FUNCTION_BLOCK AUS_FIELDBUS_USINT_TO_SIGNAL_SCALED (* Mirrors IN->OUT if Signal Valid, with scaling *)
  (* Standard: 61499-1; Description: Copyright (c) 2026 HR Agrartechnik GmbH This program and the accompanying materials are made available under the terms of the Eclipse Public License 2.0 which is available at https://www.eclipse.org/legal/epl-2.0/ SPDX-License-Identifier: EPL-2.0 *)
  (* Version 1.0, 2026-05-31, Franz Höpfinger, HR Agrartechnik GmbH *)
  PACKAGE logiBUS::signalprocessing::fieldbus;
  IMPORT eclipse4diac::core::TypeHash;
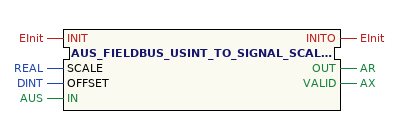
  EVENT_INPUT
    INIT : EInit; (* Init Request *)
  END_EVENT
  EVENT_OUTPUT
    INITO : EInit; (* Init Confirmation *)
  END_EVENT
  VAR_INPUT
    SCALE : REAL := REAL#1.0; (* Scaling factor *)
    OFFSET : DINT := DINT#0; (* Offset added after scaling *)
  END_VAR
  SOCKETS
    IN : adapter::types::unidirectional::AUS; (* Input *)
  END_SOCKETS
  PLUGS
    OUT : adapter::types::unidirectional::AR; (* Output Filtered *)
    VALID : adapter::types::unidirectional::AX; (* TRUE if Signal is VALID *)
  END_PLUGS
  FBS
    FIELDBUS_USINT_TO_SIGNAL_SCALED : logiBUS::signalprocessing::fieldbus::FIELDBUS_USINT_TO_SIGNAL_SCALED;
    E_D_FF : iec61499::events::E_D_FF;
  END_FBS
  EVENT_CONNECTIONS
    IN.E1 TO FIELDBUS_USINT_TO_SIGNAL_SCALED.REQ;
    FIELDBUS_USINT_TO_SIGNAL_SCALED.CNF TO OUT.E1;
    FIELDBUS_USINT_TO_SIGNAL_SCALED.CNF TO E_D_FF.CLK;
    E_D_FF.EO TO VALID.E1;
    INIT TO FIELDBUS_USINT_TO_SIGNAL_SCALED.INIT;
    FIELDBUS_USINT_TO_SIGNAL_SCALED.INITO TO INITO;
  END_CONNECTIONS
  DATA_CONNECTIONS
    IN.D1 TO FIELDBUS_USINT_TO_SIGNAL_SCALED.IN;
    FIELDBUS_USINT_TO_SIGNAL_SCALED.OUT TO OUT.D1;
    FIELDBUS_USINT_TO_SIGNAL_SCALED.VALID TO E_D_FF.D;
    E_D_FF.Q TO VALID.D1;
    SCALE TO FIELDBUS_USINT_TO_SIGNAL_SCALED.SCALE;
    OFFSET TO FIELDBUS_USINT_TO_SIGNAL_SCALED.OFFSET;
  END_CONNECTIONS
END_FUNCTION_BLOCK
